(* IEC 61131-3 sources: volt/packages/volt-lsp-iec/test-corpus/lenze-mid/Device/Plc Logic/Application/Library Manager/L_OEEA_ShiftScheduler, 3.26.4.12 (Lenze), 6 files *)

(* ---- EPROLONGBIT.dut ---- *)
TYPE EPROLONGBIT :
(
	ESHIFTDATAPROLONGED := 1,
	EPOWERONCYCLEPROLONGED := 2,
	ESHIFTDAYENDPROLONGED := 3,
	ESHIFTDAYSTARTPROLONGED := 4,
	ESHIFTDAYSTARTWAITING := 5,
	ESHIFTDAYENDWAITING := 6
);
END_TYPE

(* ---- VERSIONCONSTANTS.gvl ---- *)
VAR_GLOBAL
	GC_BYAMOUNTOFGENERALDATA : BYTE := 50;
	GC_BYAMOUNTDOWNTIMEERRORS : BYTE := 10;
	GC_IFILTERSAMPLES : INT := 20;
END_VAR

(* ---- CREATEDATETIME.pou ---- *)
FUNCTION CREATEDATETIME : DATE_AND_TIME
VAR_INPUT
	DDATE : DATE;
	TODTIME : TIME_OF_DAY;
END_VAR
END_FUNCTION

(* ---- L_OEEA_PRODUCTIONSCHEDULER.pou ---- *)
FUNCTION_BLOCK L_OEEA_PRODUCTIONSCHEDULER EXTENDS L_OEEA_Scheduler_base
VAR_INPUT
	SSHIFTNAME : STRING;
END_VAR
VAR_IN_OUT
	SCMACHINEDATA : scMachineData_base;
	SCPDPRODUCTIONDATA : scInternalProductionData;
	SCPDSHIFTDAYINDEX : scPDShiftData;
END_VAR
VAR
	RTRIGPRODSTART : R_TRIG;
	RTRIGHOLDSTART : R_TRIG;
	RTIG24EXCEEDED : R_TRIG;
	FTRIGPRODEND : F_TRIG;
	FTRIGHOLDEND : F_TRIG;
	FTRIGPOWERONDETECTED : F_TRIG;
	XPOWERONCYLCEEND : BOOL;
	XDAYENDACTIVE : BOOL;
	DTDATETIMEPREV : DATE_AND_TIME;
END_VAR
END_FUNCTION_BLOCK

(* ---- L_OEEA_SCHEDULER_BASE.pou ---- *)
FUNCTION_BLOCK L_OEEA_SCHEDULER_BASE
VAR_INPUT
	SCTRIGGER : scTrigger_base;
END_VAR
VAR_OUTPUT
	SCSHIFTVALUES : scCurrentShiftValues;
END_VAR
VAR
	EDAYOFWEEK : RTCLK.WEEKDAY;
	EDAYSTARTTIME : RTCLK.WEEKDAY;
	TONREADTIME : TON;
	UTC_HIGHRESOLUTIONTIME : SYSTIME;
	PRESULT : SysTarget.RTS_IEC_RESULT;
	LOCAL_TIME : SYSTIMEDATE;
	PEERROR : POINTER TO DTU.ERROR;
	XFIRSTPLCCYCLE : BOOL;
	XPOWERONCYCLEDETETCED : BOOL;
	XSHIFTDAYCHANGEDETECTED : BOOL;
	XSHIFTDAYSTARTDETECTED : BOOL;
	XSHIFTDAYSTARTWAITINGTIME : BOOL;
	XSHIFTDAYENDDETECTED : BOOL;
	XALLSHIFTDATAPROLONGED : BOOL;
	TONPROLONGTIMER : ARRAY [1..6] OF TON;
	FTRIGXSHIFTDAYENDPROLONGED : F_TRIG;
	FTRIGXSHIFTDAYSTARTWAITTIME : F_TRIG;
	FTRIGXPOWERONCYCLEPROLONGED : F_TRIG;
	XSHIFTDAYSTARTWAITTIMEACTIVE : BOOL;
	XSHIFTDAYCHANGEPROLONGDETECTED : BOOL;
END_VAR
END_FUNCTION_BLOCK

METHOD METH_GETDATETIME : BOOL
VAR_IN_OUT
	SCSHIFTVALUES : scCurrentShiftValues;
END_VAR
END_METHOD

METHOD METH_GETBREAKTIME : TIME
VAR_INPUT
	ESETWEEKDAY : RTCLK.WEEKDAY;
	XALLBREAKTIME : BOOL;
END_VAR
VAR_IN_OUT
	ASCDAYSCHEDULES : ARRAY [0..6] OF scDaySchedule;
END_VAR
END_METHOD

METHOD METH_PROLONGBIT : BOOL
VAR_INPUT
	TPROLONGTIME : TIME;
END_VAR
VAR_IN_OUT
	TONPROLONGTIMER : TON;
	XSTARTPROLONGTIME : BOOL;
END_VAR
END_METHOD

(* ---- L_OEEA_SHIFTSCHEDULER.pou ---- *)
FUNCTION_BLOCK L_OEEA_SHIFTSCHEDULER EXTENDS L_OEEA_Scheduler_base
VAR_INPUT
	ESHIFTMODE : enumShiftMode;
	ESETWEEKDAY : RTCLK.WEEKDAY;
	XMANUALSHIFTRESET : BOOL;
	XSHIFTPRODUCTIONACTIVE : BOOL;
	XLATERSHIFTSTARTENABLED : BOOL;
END_VAR
VAR_IN_OUT
	ASCDAYSCHEDULES : ARRAY [0..6] OF scDaySchedule;
	SCPDSHIFTDAYINDEX : scPDShiftData;
END_VAR
VAR
	EDAYOFWEEKPREVIOUS : RTCLK.WEEKDAY;
	IINDEX : INT := 1;
	JINDEX : INT := 1;
	I : INT;
	J : INT;
	K : INT;
	ISHFTCHANGECOUNTER : INT;
	XERROR : DTU.ERROR;
	XDAYCHANGEDETECTED : BOOL;
	XSHIFTCHANGEEVENTDELAY : BOOL;
	XBREAKVALID : BOOL;
	XSHIFTSTARTDETECTED : BOOL;
	TTOTALBRAKESTIME : TIME;
	INOOFBREAKSPERSHIFT : INT;
	IBREAKSHIFT : INT;
	RMINHOURDEC : REAL;
	UIMINCUT : UINT;
	RTRIGMANUALSHIFTRESET : R_TRIG;
	DTDIFFDATEANDTIME : TIME;
	DTDIFFSTARTENDTIME : TIME;
	IWEEKDAYSDIFF : INT;
	RTRIGNEWACTIVESHIFT : R_TRIG;
	FTRIGNEWACTIVESHIFT : F_TRIG;
	DTDATETIMEPRODUCTIONACTIVE : DATE_AND_TIME;
	RTRIGRODUCTIONACTIVE : R_TRIG;
	TTIMEOFSHIFTSTART : TIME;
	TTIMEOFPRODSTART : TIME;
	DTSHIFTSTART : DATE_AND_TIME;
	SDATETIMECONCAT : STRING;
	X1PLCCYCLESHIFTRESET : BOOL;
	XSETPODUCTIONACTIVE : BOOL;
	XPODUCTIONACTIVEDETECTED : BOOL;
	TODACTUALSHIFTSTARTTIME : TIME_OF_DAY;
	IACTUALSHIFT : INT;
	SCACTUALSHIFTSTARTCHANGE : scShiftSchedule;
	UIHOUR : UINT;
	UIMINUTE : UINT;
	UISECOND : UINT;
	UIMILLISECOND : UINT;
END_VAR
END_FUNCTION_BLOCK

METHOD ACT_SET_DAYSHIFTTIME
END_METHOD

METHOD ACT_SET_BREAKS
END_METHOD

METHOD ACT_FINDACTUALDAYSHIFT
END_METHOD

METHOD ACT_CALCNONPRODUCTIVETIME
END_METHOD

METHOD ACT_CREATEDAYSHIFTCHANGEEVENT
END_METHOD

METHOD ACT_STOREPDDATA
END_METHOD

METHOD ACT_POWERON
END_METHOD

METHOD ACT_SHIFTPRODACTIVE
END_METHOD
